{attribute 'qualified_only'}
{attribute 'strict'}
TYPE TaskList :
(
	IDLE, 
	HOME:=21,
	POS1, 
	POS2, 
	MOVE_UP, 
	MOVE_DOWN
)WORD;
END_TYPE

(* stored: Version 1.1.0.1, ProductVersion 3.1.4024.11
   DUT TaskList: Id {59d9b1bb-51f4-4fe9-83b4-dc92163a69c6} *)
